TYPE ST_AdaptiveModel_Output :
STRUCT
	Out1: LREAL;
END_STRUCT
END_TYPE

(* stored: Version 1.1.0.1, ProductVersion 3.1.4024.4
   DUT ST_AdaptiveModel_Output: Id {3c417d7d-04b4-4111-be11-0be255014a5c} *)
